// TIA Portal V20 export
FUNCTION "F_Safety" : Void   // FC2, LAD
{ S7_Optimized_Access := 'TRUE' }
// stored: SetENOAutomatically false
BEGIN

REGION Network 1
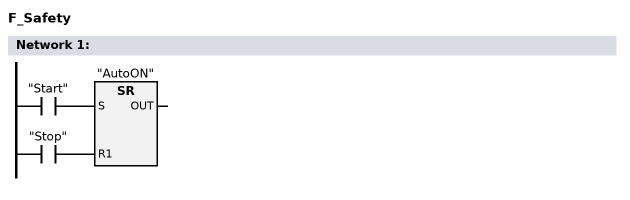
   RUNG wire#powerrail
      Contact( "Start" )
      S_SR(operand := "AutoON", r1 := wire#w1)
   END_RUNG
   RUNG wire#powerrail
      Contact( "Stop" )
   END_RUNG wire#w1
   // the same network as SCL:
   IF "Start" THEN
       "AutoON" := TRUE;   // SR flip-flop
   END_IF;
   IF "Stop" THEN "AutoON" := FALSE; END_IF;
END_REGION
END_FUNCTION
